// TIA Portal V19 export
FUNCTION "Route 404" : Void   // FC103, STL
TITLE = Polygon Transfer Line - CIP Sequence
{ S7_Optimized_Access := 'TRUE' }
// stored: AutoNumber false
   VAR_TEMP
      device_fault : Bool;
      switch_fault : Bool;
      tmp : Bool;
      Step_on : Bool;
      Dev_Check : Bool;
      New_Msg : Bool;
      Route_Ready : Bool;   // Ready to Run
      PNIOnodeFault : Bool;
      StepTime : S5Time;
      TimerError : Int;
      scratch_DI : DInt;
      scratch_Real : Real;
      Message : Int;
      scratch_I : Int;
      tmpWord : Word;
      PNIODiag : Struct
         node_2 : Struct
            failed : Bool;
            moduleFault : Bool;
         END_STRUCT;
         node_3 : Struct
            failed : Bool;
            moduleFault : Bool;
         END_STRUCT;
         node_4 : Struct
            failed : Bool;
            moduleFault : Bool;
         END_STRUCT;
         node_5 : Struct
            failed : Bool;
            moduleFault : Bool;
         END_STRUCT;
         node_6 : Struct
            failed : Bool;
            moduleFault : Bool;
         END_STRUCT;
         node_7 : Struct
            failed : Bool;
            moduleFault : Bool;
         END_STRUCT;
         node_8 : Struct
            failed : Bool;
            moduleFault : Bool;
         END_STRUCT;
         node_9 : Struct
            failed : Bool;
            moduleFault : Bool;
         END_STRUCT;
         node_10 : Struct
            failed : Bool;
            moduleFault : Bool;
            node_10 : Struct
               failed : Bool;
               moduleFault : Bool;
            END_STRUCT;
            node_11 : Struct
               failed : Bool;
               moduleFault : Bool;
               node_10 : Struct
                  failed : Bool;
                  moduleFault : Bool;
               END_STRUCT;
            END_STRUCT;
         END_STRUCT;
         node_11 : Struct
            failed : Bool;
            moduleFault : Bool;
            node_10 : Struct
               failed : Bool;
               moduleFault : Bool;
            END_STRUCT;
         END_STRUCT;
         node_12 : Struct
            failed : Bool;
            moduleFault : Bool;
            node_10 : Struct
               failed : Bool;
               moduleFault : Bool;
            END_STRUCT;
         END_STRUCT;
      END_STRUCT;
      TV_above_zero : Bool;
      TV_equal_zero : Bool;
      __PlcmigTempFillBit_38B2 : Bool;
      __PlcmigTempFillBit_38B3 : Bool;
      __PlcmigTempFillBit_38B4 : Bool;
      __PlcmigTempFillBit_38B5 : Bool;
      __PlcmigTempFillBit_38B6 : Bool;
      __PlcmigTempFillBit_38B7 : Bool;
      __PlcmigTempFillBit_39B0 : Bool;
      __PlcmigTempFillBit_39B1 : Bool;
      __PlcmigTempFillBit_39B2 : Bool;
      __PlcmigTempFillBit_39B3 : Bool;
      __PlcmigTempFillBit_39B4 : Bool;
      __PlcmigTempFillBit_39B5 : Bool;
      __PlcmigTempFillBit_39B6 : Bool;
      __PlcmigTempFillBit_39B7 : Bool;
   END_VAR
BEGIN

NETWORK
TITLE = PNIO 100 Node Faults
// PNIO Node 2
// PNIO Node 2
      A     "Module Diagnostic Result"."2_AL1103".ErrorValue.%X1;
      =     #PNIODiag.node_2.failed;
      A     "Module Diagnostic Result"."2_AL1103".ErrorValue.%X2;
      =     #PNIODiag.node_2.moduleFault;
// PNIO Node 3
      A     "Module Diagnostic Result"."3_AL1307".ErrorValue.%X1;
      =     #PNIODiag.node_3.failed;
      A     "Module Diagnostic Result"."3_AL1307".ErrorValue.%X2;
      =     #PNIODiag.node_3.moduleFault;
// PNIO Node 4
      A     "Module Diagnostic Result"."4_AL1307".ErrorValue.%X1;
      =     #PNIODiag.node_4.failed;
      A     "Module Diagnostic Result"."4_AL1307".ErrorValue.%X2;
      =     #PNIODiag.node_4.moduleFault;
// PNIO Node 5
      A     "Module Diagnostic Result"."5_AL1307".ErrorValue.%X1;
      =     #PNIODiag.node_5.failed;
      A     "Module Diagnostic Result"."5_AL1307".ErrorValue.%X2;
      =     #PNIODiag.node_5.moduleFault;
// PNIO Node 6
      A     "Module Diagnostic Result"."6_AL1307".ErrorValue.%X1;
      =     #PNIODiag.node_6.failed;
      A     "Module Diagnostic Result"."6_AL1307".ErrorValue.%X2;
      =     #PNIODiag.node_6.moduleFault;
// PNIO Node 7
      A     "Module Diagnostic Result"."7_AL1307".ErrorValue.%X1;
      =     #PNIODiag.node_7.failed;
      A     "Module Diagnostic Result"."7_AL1307".ErrorValue.%X2;
      =     #PNIODiag.node_7.moduleFault;
// PNIO Node 8
      A     "Module Diagnostic Result"."8_Promag300".ErrorValue.%X1;
      =     #PNIODiag.node_8.failed;
      A     "Module Diagnostic Result"."8_Promag300".ErrorValue.%X2;
      =     #PNIODiag.node_8.moduleFault;
// PNIO Node 9
      A     "Module Diagnostic Result"."9_SinaG120".ErrorValue.%X1;
      =     #PNIODiag.node_9.failed;
      A     "Module Diagnostic Result"."9_SinaG120".ErrorValue.%X2;
      =     #PNIODiag.node_9.moduleFault;
// PNIO Node 10
      A     "Module Diagnostic Result"."10_AL1307".ErrorValue.%X1;
      =     #PNIODiag.node_10.failed;
      A     "Module Diagnostic Result"."10_AL1307".ErrorValue.%X2;
      =     #PNIODiag.node_10.moduleFault;
// PNIO Node 11
      A     "Module Diagnostic Result"."11_PNCoup".ErrorValue.%X1;
      =     #PNIODiag.node_11.failed;
      A     "Module Diagnostic Result"."11_PNCoup".ErrorValue.%X2;
      =     #PNIODiag.node_11.moduleFault;
// PNIO Node 12
      A     "Module Diagnostic Result"."12_AL1307".ErrorValue.%X1;
      =     #PNIODiag.node_12.failed;
      A     "Module Diagnostic Result"."12_AL1307".ErrorValue.%X2;
      =     #PNIODiag.node_12.moduleFault;


NETWORK
TITLE = PNIO node fault
      O     #PNIODiag.node_2.failed;
      O     #PNIODiag.node_2.moduleFault;
      O     #PNIODiag.node_3.failed;
      O     #PNIODiag.node_3.moduleFault;
      O     #PNIODiag.node_4.failed;
      O     #PNIODiag.node_4.moduleFault;
      O     #PNIODiag.node_5.failed;
      O     #PNIODiag.node_5.moduleFault;
      O     #PNIODiag.node_6.failed;
      O     #PNIODiag.node_6.moduleFault;
      O     #PNIODiag.node_7.failed;
      O     #PNIODiag.node_7.moduleFault;
      O     #PNIODiag.node_8.failed;
      O     #PNIODiag.node_8.moduleFault;
      O     #PNIODiag.node_9.failed;
      O     #PNIODiag.node_9.moduleFault;
      O     #PNIODiag.node_10.failed;
      O     #PNIODiag.node_10.moduleFault;
      O     #PNIODiag.node_11.failed;
      O     #PNIODiag.node_11.moduleFault;
      O     #PNIODiag.node_12.failed;
      O     #PNIODiag.node_12.moduleFault;
      =     #PNIOnodeFault;

NETWORK
TITLE = Device Faults
      O     "ItemAlarmsOP".Item[20];  //FB_FAULT_VALVE_09_05
      O     "ItemAlarmsOP".Item[23];  //FB_FAULT_VALVE_09_08
      O     "ItemAlarmsOP".Item[24];  //FB_FAULT_VALVE_09_09
      O     "ItemAlarmsOP".Item[25];  //FB_FAULT_VALVE_09_10
      O     "ItemAlarmsOP".Item[26];  //FB_FAULT_VALVE_09_11
      O     "ItemInfoScada".Items[68].fb_error;
      O     "ItemInfoScada".Items[69].fb_error;
      O     "ItemInfoScada".Items[70].fb_error;
      O     "ItemInfoScada".Items[85].fb_error;
      O     "ItemInfoScada".Items[71].fb_error;
      O     "ItemInfoScada".Items[72].fb_error;
      O     "ItemInfoScada".Items[73].fb_error;
      O     "ItemInfoScada".Items[74].fb_error;
      O     "ItemInfoScada".Items[78].fb_error;
      O     "ItemInfoScada".Items[79].fb_error;
      O     "ItemInfoScada".Items[80].fb_error;
      O     "ItemInfoScada".Items[81].fb_error;
      O     "ItemInfoScada".Items[82].fb_error;
      O     "ItemInfoScada".Items[83].fb_error;
      O     "ItemInfoScada".Items[75].fb_error;
      O     "ItemInfoScada".Items[76].fb_error;
      O     "ItemInfoScada".Items[77].TrippedInd;
      O     "ItemInfoScada".Items[77].IsolatedInd;
      O     "ItemInfoScada".Items[84].TrippedInd;
      O     "ItemInfoScada".Items[84].IsolatedInd;
      O     "ItemInfoScada".Items[77].fb_error;
      O     "ItemInfoScada".Items[84].fb_error;
      O     #PNIOnodeFault;
      O     "ProcessAndPbAlarms"."A"[78];  //A78_PG_PTX0940HighPress
      O     "ProcessAndPbAlarms"."A"[69];  //A69_TT0941_TempFault
      =     #device_fault;

NETWORK
TITLE = Switch Fault
      ON    "PG_Devices".DI_100_005_X06_X1_3p4;
      O     "PG_Devices".DI_100_005_X06_X1_3p2;
      O     "PG_Devices".DI_100_012_X1_1p2;
      =     #switch_fault;

NETWORK
TITLE = Set Devices in Auto
      A     "RTE_404_DB".HMI.RUNNING;
      R     "ItemInfoScada".Items[50].auto_man;
      R     "ItemInfoScada".Items[53].auto_man;
      R     "ItemInfoScada".Items[54].auto_man;
      R     "ItemInfoScada".Items[55].auto_man;
      R     "ItemInfoScada".Items[56].auto_man;
      R     "ItemInfoScada".Items[76].auto_man;
      R     "ItemInfoScada".Items[78].auto_man;
      R     "ItemInfoScada".Items[79].auto_man;
      R     "ItemInfoScada".Items[80].auto_man;
      R     "ItemInfoScada".Items[81].auto_man;
      R     "ItemInfoScada".Items[82].auto_man;
      R     "ItemInfoScada".Items[83].auto_man;
      R     "ItemInfoScada".Items[77].auto_man;
      R     "ItemInfoScada".Items[84].auto_man;

NETWORK
TITLE = Route Healthy
      AN    #device_fault;
      AN    #switch_fault;
      =     "RTE_404_DB".HMI.Route_Healthy;

NETWORK
TITLE = DEVICE FAULT STATUS
      A     #device_fault;
      AN    "RTE_404_TestBit";
      =     "RTE_404_DB".FLAGS.Device_Fault;

NETWORK
TITLE = GENERAL FAULT STATUS
      O     #switch_fault;
      O     "RTE_404_DB".FLAGS.Device_Fault;
      A     "RTE_404_DB".HMI.RUNNING;
      =     "RTE_404_DB".HMI.FAULT;

NETWORK
TITLE = Temporary Message Store
// Clear down temporary message store.
      L     0;
      T     #Message;
      NOP   0;

NETWORK
TITLE = Generate Sequence Start Command
// The sequence is initiated via the interface signals ..afl
      A     "RTE_404_DB".HMI_CMD.Start;
      AN    "RTE_404_DB".HMI.RUNNING;
      A     "RTE_404_DB".HMI.Route_Healthy;
      =     "RTE_404_DB".FLAGS.Sequence_Start;


      A     "RTE_404_DB".HMI_CMD.Start;
      A     "RTE_404_DB".HMI.SEQUENCE_ABORTED;
      JCN   a10a;
      L     0;
      T     "RTE_404_DB".HMI.NEXT_STEP;
a10a: NOP   0;

      AN    "RTE_404_DB".HMI.RUNNING;
      A     "RTE_404_DB".HMI.Route_Healthy;
      =     "RTE_404_DB".HMI_CMD.Start_Available;


NETWORK
TITLE = ****ERROR MESSAGE****
// Message 10 - Device Fault
      A(;
      O     "RTE_404_DB".HMI_CMD.Start;
      O     "RTE_404_DB".HMI_CMD.Continue;
      );
      A     #device_fault;
      JNB   _001;
      L     10;
      T     #Message;
      SET;
      SAVE;
      CLR;
_001: A     BR;
      JC    AA01;

NETWORK
TITLE = ****ERROR MESSAGE****
// Message 12 - Control Stop activated
      A(;
      O     "RTE_404_DB".HMI_CMD.Start;
      O     "RTE_404_DB".HMI_CMD.Continue;
      );
      A(;
      O     "PG_Devices".DI_100_012_X1_1p2;
      O;
      A     "RTE_404_DB".FLAGS.STEP_4_0;
      AN    "CIP_Running";
      );
      JNB   _002;
      L     41;
      T     #Message;
      SET;
      SAVE;
      CLR;
_002: A     BR;
      JC    AA01;

NETWORK
TITLE = ****ERROR MESSAGE****
// Message 37 - Swingbend out of position
      A(;
      O     "RTE_404_DB".HMI_CMD.Start;
      O     "RTE_404_DB".HMI_CMD.Continue;
      );
      A(;
      O     "PG_Devices".DI_100_005_X06_X1_3p2;
      ON    "PG_Devices".DI_100_005_X06_X1_3p4;
      );
      JNB   _003;
      L     37;
      T     #Message;
      SET;
      SAVE;
      CLR;
_003: A     BR;
      JC    AA01;

NETWORK
TITLE = ****ERROR MESSAGE****
// Message 17 - Sequence Not Held
// To abort or continue the clean it must have already been held.
      A(;
      O     "RTE_404_DB".HMI_CMD.Abort;
      O     "RTE_404_DB".HMI_CMD.Continue;
      );
      AN    "RTE_404_DB".HMI.SEQUENCE_HELD;
      JNB   _004;
      L     17;
      T     #Message;
      SET;
      SAVE;
      CLR;
_004: A     BR;
      JC    AA01;

NETWORK
TITLE = ****ERROR MESSAGE****
// Message 21 - Line Sterilising
// *** Use Sterilising Seq running bit ***
      A(;
      O     "RTE_404_DB".HMI_CMD.Start;
      O     "RTE_404_DB".HMI_CMD.Continue;
      );
      A     "ATI";
      AN    "ATI";
      JNB   _005;
      L     21;
      T     #Message;
      SET;
      SAVE;
      CLR;
_005: A     BR;
      JC    AA01;

NETWORK
TITLE = ****ERROR MESSAGE****
// Message 22 - Inhibited by Running Sequence
// *** Use Production Seq running bit ***
      A(;
      O     "RTE_404_DB".HMI_CMD.Start;
      O     "RTE_404_DB".HMI_CMD.Continue;
      );
      A(;
      O     "RTE_405_DB".HMI.RUNNING;
      O     "RTE_406_DB".HMI.RUNNING;
      );
      JNB   _006;
      L     22;
      T     #Message;
      SET;
      SAVE;
      CLR;
_006: A     BR;
      JC    AA01;

NETWORK
TITLE = ****ERROR MESSAGE****
// Message 25 - CIP Not Running
      A(;
      O     "RTE_404_DB".HMI_CMD.Start;
      O     "RTE_404_DB".HMI_CMD.Continue;
      );
      A     "RTE_404_DB".FLAGS.STEP_4_0;
      AN    "CIP_Running";
      JNB   _007;
      L     25;
      T     #Message;
      SET;
      SAVE;
      CLR;
_007: A     BR;
      JC    AA01;

NETWORK
TITLE = New Message Detected
AA01: A(;
      L     #Message;
      L     0;
      <>I;
      );
      JNB   _008;
      L     #Message;
      T     "RTE_404_DB".HMI.ERROR_TEXT_NUMBER;
      SET;
      SAVE;
      CLR;
_008: A     BR;
      =     #New_Msg;

NETWORK
TITLE = ****NEW ERROR MESSAGE****
// Reset all CIP commands except START.
// On a new non-zero error message being displayed reset all commands from SCADA 
// so they take no action. Also, start a delay off timer to cancel display of the 
// error message.
      A     #New_Msg;
      R     "RTE_404_DB".HMI_CMD.Abort;
      R     "RTE_404_DB".HMI_CMD.Continue;
      R     "RTE_404_DB".HMI_CMD.Hold;
      R     "RTE_404_DB".HMI_CMD.Timer_Release;
      R     "RTE_404_DB".HMI_CMD.Timer_Hold;
      R     "RTE_404_DB".FLAGS.Sequence_Start;
      L     S5T#10S;
      SF    "RTE404_MSG";

NETWORK
TITLE = ****NEW ERROR MESSAGE****
// Error message display cancel.
      AN    "RTE404_MSG";
      JNB   _009;
      L     0;
      T     "RTE_404_DB".HMI.ERROR_TEXT_NUMBER;
_009: NOP   0;

NETWORK
TITLE = ROUTE RUNNING
      L     "RTE_404_DB".HMI.STEP_NUMBER;
      L     0;
      <>I;
      =     "RTE_404_DB".HMI.RUNNING;

NETWORK
TITLE = ****SEQ ABORT****
      A     "RTE_404_DB".HMI_CMD.Abort;
      A     "RTE_404_DB".HMI.SEQUENCE_HELD;
      S     "RTE_404_DB".HMI.SEQUENCE_ABORTED;

      A     "RTE_404_DB".HMI.SEQUENCE_HELD;
      =     "RTE_404_DB".HMI_CMD.Abort_Available;


NETWORK
TITLE = Enable HMI Hold Pb
      A     "RTE_404_DB".HMI.RUNNING;
      =     "RTE_404_DB".HMI_CMD.Hold_Available;

NETWORK
TITLE = Sequence held flag
// Set sequence hold if sequence is running and a hold fault condition is detected 
// or a sequence hold command is received from SCADA.
// 
// When a validated CONTINUE command is received from SCADA and all fault 
// conditions are cleared then reset sequence hold.
// 
// Added "Product Request" (CIP Complete) to prevent sequence going into hold when 
// Central CIP completes
      A(;
      O     "RTE_404_DB".HMI_CMD.Hold;
      ON    "RTE_404_DB".HMI.Route_Healthy;
      O;
      A(;
      O     "RTE_404_DB".FLAGS.STEP_3_0;
      O     "RTE_404_DB".FLAGS.STEP_4_0;
      );
      AN    "Product_Request";
      AN    "CIP_Running";
      );
      A     "RTE_404_DB".HMI.RUNNING;
      =     #__PlcmigTempFillBit_39B0;
      A     #__PlcmigTempFillBit_39B0;
      BLD   102;
      S     "RTE_404_DB".HMI.SEQUENCE_HELD;
      A     #__PlcmigTempFillBit_39B0;
      NOT;
      =     #__PlcmigTempFillBit_39B1;
      A     #__PlcmigTempFillBit_39B1;
      A(;
      O     "RTE_404_DB".HMI_CMD.Continue;
      O     "RTE_404_DB".HMI_CMD.Abort;
      );
      R     "RTE_404_DB".HMI.SEQUENCE_HELD;
      A     #__PlcmigTempFillBit_39B1;
      A     "RTE_404_DB".HMI.SEQUENCE_HELD;
      =     "RTE_404_DB".HMI_CMD.Continue_Available;

NETWORK
TITLE = Sequence held flag
// Reset when circuit not running i.e after an abort.
      A     "RTE_404_DB".FLAGS.STEP_0;
      AN    "RTE_404_DB".HMI.RUNNING;
      R     "RTE_404_DB".HMI.SEQUENCE_HELD;

NETWORK
TITLE = ****RESET ABORT FLAG****
      A     "RTE_404_DB".FLAGS.STEP_0;
      A     "RTE_404_DB".FLAGS.Step_Change;
      R     "RTE_404_DB".HMI.SEQUENCE_ABORTED;

NETWORK
TITLE = Step 0.0 Reset
      AN    "RTE_404_DB".HMI.RUNNING;
      AN    "RTE_404_DB".FLAGS.STEP_0;
      =     #Step_on;

NETWORK
TITLE = Step 0.0 Reset
// Reset sequnece to step 0 and clear down step value and dimension words.
      A(;
      A(;
      A(;
      O     #Step_on;
      O;
      A     "RTE_404_DB".FLAGS.STEP_0;
      A     "RTE_404_DB".FLAGS.Step_Change;
      );
      JNB   _00a;
      L     0;
      T     "RTE_404_DB".HMI.NEXT_STEP;
      SET;
      SAVE;
      CLR;
_00a: A     BR;
      );
      JNB   _00b;
      L     0;
      T     "RTE_404_DB".HMI.STEP_VALUE;
      SET;
      SAVE;
      CLR;
_00b: A     BR;
      );
      JNB   _00c;
      L     0;
      T     "RTE_404_DB".HMI.STEP_VALUE_DIMENSION;
_00c: NOP   0;

NETWORK
TITLE = Move to Step 0.5
      A     "RTE_404_DB".FLAGS.STEP_0;
      A     "RTE_404_DB".FLAGS.Sequence_Start;
      =     #__PlcmigTempFillBit_39B0;
      A     #__PlcmigTempFillBit_39B0;
      BLD   102;
      =     #Step_on;
      A     #__PlcmigTempFillBit_39B0;
      JNB   _00d;
      L     5;
      T     "RTE_404_DB".HMI.NEXT_STEP;
_00d: NOP   0;

NETWORK
TITLE = Set Line Status Unsterile
      A     #Step_on;
      R     "RTE_404_DB".FLAGS.Clean;
      R     "RTE_405_DB".FLAGS.Sterile;

NETWORK
TITLE = Move to Step 1.0
      A(;
      L     "RTE_404_DB".HMI.NEXT_STEP;
      L     5;
      ==I;
      );
      A     "CIP_Route_Request";
      AN    "RTE_404_DB".FLAGS.Step_Change;
      =     #__PlcmigTempFillBit_39B0;
      A     #__PlcmigTempFillBit_39B0;
      BLD   102;
      =     #Step_on;
      A     #__PlcmigTempFillBit_39B0;
      JNB   _00e;
      L     10;
      T     "RTE_404_DB".HMI.NEXT_STEP;
_00e: NOP   0;

NETWORK
TITLE = Dev Check
// Dev Check following Route valves Open - 09.10, 09.08, 09.45, 10.21, 10.23, 10.25
// and following Route Valves closed - 09.09, 09.05, 10.24
      A     "RTE_404_DB".FLAGS.STEP_1_0;
      A     "Y0905R";
      A     "Y0908S";
      A     "Y0909R";
      A     "Y0910S";
      A(;
      A     "ItemInfoScada".Items[78].Set_FB;
      A     "ItemInfoScada".Items[79].Set_FB;
      A     "ItemInfoScada".Items[80].Reset_FB;
      );
      =     #Dev_Check;

NETWORK
TITLE = Move to Step 2.0
      A     "RTE_404_DB".FLAGS.STEP_1_0;
      A     #Dev_Check;
      AN    "RTE_404_DB".FLAGS.Step_Change;
      =     #__PlcmigTempFillBit_39B0;
      A     #__PlcmigTempFillBit_39B0;
      BLD   102;
      =     #Step_on;
      A     #__PlcmigTempFillBit_39B0;
      JNB   _00f;
      L     20;
      T     "RTE_404_DB".HMI.NEXT_STEP;
_00f: NOP   0;

NETWORK
TITLE = Check Condenstate OK, then Set CIP Route Open
      A     "RTE_404_DB".FLAGS.STEP_2_0;
      A     "CIP_Route_Request";
      A     "M21.2";
      S     "RTE_404_Cip_Route_Open";

NETWORK
TITLE = Move to Step 3.0
      A     "RTE_404_DB".FLAGS.STEP_2_0;
      A     "CIP_Running";
      AN    "RTE_404_DB".FLAGS.Step_Change;
      =     #__PlcmigTempFillBit_39B0;
      A     #__PlcmigTempFillBit_39B0;
      BLD   102;
      =     #Step_on;
      A     #__PlcmigTempFillBit_39B0;
      JNB   _010;
      L     30;
      T     "RTE_404_DB".HMI.NEXT_STEP;
_010: NOP   0;

NETWORK
TITLE = Reset Totaliser Value
// Totaliser Control
// 0 = Totalise
// 3 = Reset + Totalise
      O(;
      A(;
      A(;
      O     "RTE_404_DB".FLAGS.STEP_3_0;
      O;
      AN    "M21.2";
      A     "RTE_404_DB".FLAGS.STEP_4_0;
      );
      =     "RTE_404_Sip_Steam";
      A     "RTE_404_Sip_Steam";
      JNB   _011;
      L     "RTE_404_DB".PARAMETERS.PARAM_01;
      ITD;
      T     #scratch_DI;
      SET;
      SAVE;
      CLR;
_011: A     BR;
      );
      JNB   _012;
      L     #scratch_DI;
      DTR;
      T     #scratch_Real;
      SET;
      SAVE;
      CLR;
_012: A     BR;
      );
      O(;
      A(;
      O     #Step_on;
      O;
      A     "RTE_404_DB".FLAGS.STEP_3_0;
      A(;
      O     #device_fault;
      ON    "CIP_Running";
      );
      );
      A(;
      L     "PG_Devices".FT0940.Totaliser_Value;
      L     0.0;
      <>R;
      );
      =     #TV_above_zero;
      A     #TV_above_zero;
      JNB   _013;
      L     1;
      T     "PG_Devices".FT0940.Totaliser_Control;
      SET;
      SAVE;
      CLR;
_013: A     BR;
      );
      O(;
      A(;
      A     "RTE_404_DB".FLAGS.STEP_3_0;
      A(;
      L     "PG_Devices".FT0940.Totaliser_Value;
      L     0.0;
      <=R;
      );
      JNB   _014;
      L     0;
      T     "PG_Devices".FT0940.Totaliser_Control;
      SET;
      SAVE;
      CLR;
_014: A     BR;
      );
      =     #TV_equal_zero;
      A     #TV_equal_zero;
      );
      O(;
      A     #TV_above_zero;
      S     "RTE_404_DB".FLAGS.TotaliserResetBit;
      A     #TV_equal_zero;
      R     "RTE_404_DB".FLAGS.TotaliserResetBit;
      A     "RTE_404_DB".FLAGS.TotaliserResetBit;
      );
      =     #tmp;

NETWORK
TITLE = Move to Step 4.0
      AN    "RTE_404_DB".FLAGS.TotaliserResetBit;
      A     "RTE_404_DB".FLAGS.STEP_3_0;
      A(;
      L     "PG_Devices".FT0940.Totaliser_Value;
      L     #scratch_Real;
      >=R;
      );
      AN    "RTE_404_DB".FLAGS.Step_Change;
      =     #__PlcmigTempFillBit_39B0;
      A     #__PlcmigTempFillBit_39B0;
      BLD   102;
      =     #Step_on;
      A     #__PlcmigTempFillBit_39B0;
      JNB   _015;
      L     40;
      T     "RTE_404_DB".HMI.NEXT_STEP;
_015: NOP   0;

NETWORK
TITLE = EOL Valve Flips Interval Timer
      A     "RTE_404_DB".FLAGS.STEP_4_0;
      AN    "RTE_404_DB".FLAGS.ENCYL_3;
      AN    "RTE_404_DB".HMI.SEQUENCE_HELD;
      =     #__PlcmigTempFillBit_39B0;
      BLD   103;
      A     "RTE_404_DB".FLAGS.ENCYL_3;
      =     #__PlcmigTempFillBit_39B1;
      BLD   103;
      A(;
      A(;
      L     "RTE_404_DB".PARAMETERS.PARAM_03;
      ITD;
      T     #scratch_DI;
      SET;
      SAVE;
      CLR;
      A     BR;
      );
      JNB   _016;
      L     #scratch_DI;
      L     1000;
      *D;
      T     #scratch_DI;
      AN    OV;
      SAVE;
      CLR;
_016: A     BR;
      );
      JNB   _017;
      CALL  "TONR"
      ( TMR_EN  := #__PlcmigTempFillBit_39B0,
        RESET   := #__PlcmigTempFillBit_39B1,
        PV      := #scratch_DI,
        DELTA_T := "Last Scan Time",
        Q       := "RTE_404_DB".FLAGS.ENCYL_1,
        ET      := "RTE_404_DB".PARAMETERS.PARAM_03_Act
      );
_017: NOP   0;

NETWORK
TITLE = Cycle 1 to Cycle 2 Delay Timer.
      A     "RTE_404_DB".FLAGS.STEP_4_0;
      A     "RTE_404_DB".FLAGS.ENCYL_1;
      AN    "RTE_404_DB".HMI.SEQUENCE_HELD;
      =     #__PlcmigTempFillBit_39B0;
      BLD   103;
      AN    "RTE_404_DB".FLAGS.ENCYL_1;
      =     #__PlcmigTempFillBit_39B1;
      BLD   103;
      A(;
      A(;
      L     "RTE_404_DB".PARAMETERS.PARAM_04;
      ITD;
      T     #scratch_DI;
      SET;
      SAVE;
      CLR;
      A     BR;
      );
      JNB   _018;
      L     #scratch_DI;
      L     1000;
      *D;
      T     #scratch_DI;
      AN    OV;
      SAVE;
      CLR;
_018: A     BR;
      );
      JNB   _019;
      CALL  "TONR"
      ( TMR_EN  := #__PlcmigTempFillBit_39B0,
        RESET   := #__PlcmigTempFillBit_39B1,
        PV      := #scratch_DI,
        DELTA_T := "Last Scan Time",
        Q       := "RTE_404_DB".FLAGS.ENCYL_2,
        ET      := "RTE_404_DB".PARAMETERS.PARAM_04_Act
      );
_019: NOP   0;

NETWORK
TITLE = Cycle 2 to Cycle 3 Overlapping Timers.
      A     "RTE_404_DB".FLAGS.STEP_4_0;
      A     "RTE_404_DB".FLAGS.ENCYL_2;
      =     #__PlcmigTempFillBit_39B0;
      A     #__PlcmigTempFillBit_39B0;
      L     S5T#2S;
      SD    "Tag_78";
      NOP   0;
      NOP   0;
      NOP   0;
      NOP   0;
      A     #__PlcmigTempFillBit_39B0;
      BLD   102;
      L     S5T#2S;
      SF    "T83";

NETWORK
TITLE = Cycle 2 + T69 (2 Secs) to Cycle 3 Delay Timer.
      A     "RTE_404_DB".FLAGS.STEP_4_0;
      A     "RTE_404_DB".FLAGS.ENCYL_2;
      A     "Tag_78";
      AN    "RTE_404_DB".HMI.SEQUENCE_HELD;
      =     #__PlcmigTempFillBit_39B0;
      BLD   103;
      AN    "RTE_404_DB".FLAGS.ENCYL_2;
      =     #__PlcmigTempFillBit_39B1;
      BLD   103;
      A(;
      A(;
      L     "RTE_404_DB".PARAMETERS.PARAM_05;
      ITD;
      T     #scratch_DI;
      SET;
      SAVE;
      CLR;
      A     BR;
      );
      JNB   _01a;
      L     #scratch_DI;
      L     1000;
      *D;
      T     #scratch_DI;
      AN    OV;
      SAVE;
      CLR;
_01a: A     BR;
      );
      JNB   _01b;
      CALL  "TONR"
      ( TMR_EN  := #__PlcmigTempFillBit_39B0,
        RESET   := #__PlcmigTempFillBit_39B1,
        PV      := #scratch_DI,
        DELTA_T := "Last Scan Time",
        Q       := "RTE_404_DB".FLAGS.ENCYL_3,
        ET      := "RTE_404_DB".PARAMETERS.PARAM_05_Act
      );
_01b: NOP   0;

NETWORK
TITLE = Move to Step 5.0
// Product_Request means "CIP Complete" in this context.
      A(;
      A     "RTE_404_DB".FLAGS.STEP_4_0;
      A     "Product_Request";
      O;
      A     "RTE_404_DB".HMI_CMD.Abort;
      A     "RTE_404_DB".HMI.SEQUENCE_ABORTED;
      );
      AN    "RTE_404_DB".FLAGS.Step_Change;
      =     #__PlcmigTempFillBit_39B0;
      A     #__PlcmigTempFillBit_39B0;
      BLD   102;
      =     #Step_on;
      A     #__PlcmigTempFillBit_39B0;
      JNB   _01c;
      L     50;
      T     "RTE_404_DB".HMI.NEXT_STEP;
_01c: NOP   0;

NETWORK
TITLE = Move to Step 6.0
      A     "RTE_404_DB".FLAGS.STEP_5_0;
      A     "Y0910R";
      =     #__PlcmigTempFillBit_39B0;
      A     #__PlcmigTempFillBit_39B0;
      AN    "RTE_404_DB".FLAGS.Step_Change;
      =     #__PlcmigTempFillBit_39B1;
      A     #__PlcmigTempFillBit_39B1;
      BLD   102;
      =     #Step_on;
      A     #__PlcmigTempFillBit_39B1;
      JNB   _01d;
      L     60;
      T     "RTE_404_DB".HMI.NEXT_STEP;
_01d: NOP   0;
      A     #__PlcmigTempFillBit_39B0;
      BLD   102;
      R     "RTE_404_Cip_Route_Open";

NETWORK
TITLE = Dev Check
// Check following valve are open  V09.11, V10.25, V10.27, V10.83
      A     "RTE_404_DB".FLAGS.STEP_6_0;
      A     "Y0908S";
      A     "Y0910R";
      A     "Y0911S";
      A(;
//   A     "ItemInfoScada".items[79].Set_FB
      A     "ItemInfoScada".Items[81].Set_FB;
      A     "ItemInfoScada".Items[82].Set_FB;
      A     "ItemInfoScada".Items[83].Set_FB;
      );
      =     #Dev_Check;

NETWORK
TITLE = Move to Step 7.0
      A     "RTE_404_DB".FLAGS.STEP_6_0;
      A     #Dev_Check;
      AN    "RTE_404_DB".FLAGS.Step_Change;
      =     #__PlcmigTempFillBit_39B0;
      A     #__PlcmigTempFillBit_39B0;
      BLD   102;
      =     #Step_on;
      A     #__PlcmigTempFillBit_39B0;
      JNB   _01e;
      L     70;
      T     "RTE_404_DB".HMI.NEXT_STEP;
_01e: NOP   0;

NETWORK
TITLE = Initialise Step Parameters
      A(;
      A     #Step_on;
      JNB   _01f;
      L     "RTE_404_DB".PARAMETERS.PARAM_02;
      T     "RTE_404_DB".HMI.STEP_VALUE;
      SET;
      SAVE;
      CLR;
_01f: A     BR;
      );
      JNB   _020;
      L     1;
      T     "RTE_404_DB".HMI.STEP_VALUE_DIMENSION;
_020: NOP   0;

NETWORK
TITLE = Move to Step 8.0
      A     "RTE_404_DB".FLAGS.STEP_7_0;
      A     "RTE_404_DB".FLAGS.Step_Value_Done;
      AN    "RTE_404_DB".FLAGS.Step_Change;
      =     #__PlcmigTempFillBit_39B0;
      A     #__PlcmigTempFillBit_39B0;
      BLD   102;
      =     #Step_on;
      A     #__PlcmigTempFillBit_39B0;
      JNB   _021;
      L     80;
      T     "RTE_404_DB".HMI.NEXT_STEP;
_021: NOP   0;

NETWORK
TITLE = Dev Check
// V09.11
//     V09.08
//     V10.21
//     V10.23
//     V10.27
//     V10.83
//     V10.25
      A     "Y0908R";
      A     "Y0911R";
      A     "ItemInfoScada".Items[78].Reset_FB;
      A     "ItemInfoScada".Items[79].Reset_FB;
      A     "ItemInfoScada".Items[81].Reset_FB;
      A     "ItemInfoScada".Items[82].Reset_FB;
      A     "ItemInfoScada".Items[83].Reset_FB;
      =     #Dev_Check;

NETWORK
TITLE = Move to Step END
      A     "RTE_404_DB".FLAGS.STEP_8_0;
      A     #Dev_Check;
      AN    "RTE_404_DB".FLAGS.Step_Change;
      =     #__PlcmigTempFillBit_39B0;
      A     #__PlcmigTempFillBit_39B0;
      BLD   102;
      =     #Step_on;
      A     #__PlcmigTempFillBit_39B0;
      JNB   _022;
      L     90;
      T     "RTE_404_DB".HMI.NEXT_STEP;
_022: NOP   0;

NETWORK
TITLE = Set Line Status Unsterile
      A     #Step_on;
      AN    "RTE_404_DB".HMI.SEQUENCE_ABORTED;
      S     "RTE_404_DB".FLAGS.Clean;

NETWORK
TITLE = Move to Step 0.0
      A     "RTE_404_DB".FLAGS.STEP_END;
      A     "RTE_404_DB".FLAGS.Step_Value_Done;
      AN    "RTE_404_DB".FLAGS.Step_Change;
      =     #__PlcmigTempFillBit_39B0;
      A     #__PlcmigTempFillBit_39B0;
      BLD   102;
      =     #Step_on;
      A     #__PlcmigTempFillBit_39B0;
      JNB   _023;
      L     0;
      T     "RTE_404_DB".HMI.NEXT_STEP;
_023: NOP   0;

NETWORK
TITLE = Step Change Detected
// The next step number is different to the current step then set flag.
      L     "RTE_404_DB".HMI.NEXT_STEP;
      L     "RTE_404_DB".HMI.STEP_NUMBER;
      <>I;
      =     "RTE_404_DB".FLAGS.Step_Change;

NETWORK
TITLE = Current step value decremented to zero
      A(;
      L     "RTE_404_DB".HMI.STEP_VALUE;
      L     0;
      <=I;
      );
      AN    "RTE_404_DB".FLAGS.Step_Change;
      =     "RTE_404_DB".FLAGS.Step_Value_Done;

NETWORK
TITLE = Enable step count down
      A(;
      A     "RTE_404_DB".FLAGS.STEP_7_0;
      A(;
      ON    "Y0908S";
      ON    "Y0910R";
      ON    "Y0911S";
      ON    "ItemInfoScada".Items[79].Set_FB;
      ON    "ItemInfoScada".Items[81].Set_FB;
      ON    "ItemInfoScada".Items[82].Set_FB;
      ON    "ItemInfoScada".Items[83].Set_FB;
      );
      O     "RTE_404_DB".HMI.SEQUENCE_HELD;
      );
      NOT;
      =     "RTE_404_DB".FLAGS.Step_Count_Enable;

NETWORK
TITLE = Decrement Step Value
// With count enabled and timer not held count down on each 1 second pulse.
      A     "RTE_404_DB".HMI.RUNNING;
      A     "RTE_404_DB".FLAGS.Step_Count_Enable;
      AN    "RTE_404_DB".HMI.TIMER_HELD;
      AN    "RTE_404_DB".FLAGS.Step_Value_Done;
      A     "1HZ_ONESHOT";
      JNB   _024;
      L     "RTE_404_DB".HMI.STEP_VALUE;
      L     1;
      -I;
      T     "RTE_404_DB".HMI.STEP_VALUE;
_024: NOP   0;

NETWORK
TITLE = Reset HMI commands
      A     "ATI";
      R     "RTE_404_DB".HMI_CMD.Abort;
      R     "RTE_404_DB".HMI_CMD.Continue;
      R     "RTE_404_DB".HMI_CMD.Hold;
      R     "RTE_404_DB".HMI_CMD.Timer_Release;
      R     "RTE_404_DB".HMI_CMD.Timer_Hold;
      R     "RTE_404_DB".HMI_CMD.Start;

NETWORK
TITLE = MESSAGE CLEARANCE TIMING
      A     "1HZ_ONESHOT";
      =     #__PlcmigTempFillBit_39B0;
      BLD   103;
      CALL  "ERROR_MSG_CLEAR"
      ( MESSAGE_CLEAR_TIME := 10,
        SECOND_PULSE       := #__PlcmigTempFillBit_39B0,
        ERROR_MESSAGE      := "RTE_404_DB".HMI.ERROR_TEXT_NUMBER,
        ERROR_MESSAGE_MEM  := "RTE_404_DB".CONTROL.ERROR_MESSAGE_MEM,
        ELAPSED_TIME       := "RTE_404_DB".CONTROL.MESSAGE_TIME
      );
      NOP   0;

NETWORK
TITLE = STEP TIMER
// On detection of a new step, the timer is reset to 0 and will then start timing 
// whilst on the current step.
      A     "1HZ_ONESHOT";
      =     #__PlcmigTempFillBit_39B0;
      BLD   103;
      CALL  "STEP_TIMER"
      ( DBNR                   := 404,
        NEXT_STEP_LOCATION     := 18,
        STEP_NUM_LOCATION      := 2,
        TIME_PULSE             := #__PlcmigTempFillBit_39B0,
        STEP_TIME_ACC_LOCATION := 26
      );
      NOP   0;

NETWORK
TITLE = 
      A     "RTE_404_DB".FLAGS.Step_Change;
      JNB   _025;
      L     "RTE_404_DB".HMI.NEXT_STEP;
      T     "RTE_404_DB".HMI.STEP_NUMBER;
_025: NOP   0;

NETWORK
TITLE = Spare
      L     "RTE_404_DB".HMI.STEP_NUMBER;
      L     0;
      ==I;
      =     "RTE_404_DB".FLAGS.STEP_0;

NETWORK
TITLE = Spare
      O     "RTE_404_DB".HMI.RUNNING;
      ON    "RTE_404_DB".HMI.RUNNING;
      =     #__PlcmigTempFillBit_39B0;
      A     #__PlcmigTempFillBit_39B0;
      A(;
      L     "RTE_404_DB".HMI.STEP_NUMBER;
      L     10;
      ==I;
      );
      =     "RTE_404_DB".FLAGS.STEP_1_0;
      A     #__PlcmigTempFillBit_39B0;
      A(;
      L     "RTE_404_DB".HMI.STEP_NUMBER;
      L     20;
      ==I;
      );
      =     "RTE_404_DB".FLAGS.STEP_2_0;
      A     #__PlcmigTempFillBit_39B0;
      A(;
      L     "RTE_404_DB".HMI.STEP_NUMBER;
      L     30;
      ==I;
      );
      =     "RTE_404_DB".FLAGS.STEP_3_0;
      A     #__PlcmigTempFillBit_39B0;
      A(;
      L     "RTE_404_DB".HMI.STEP_NUMBER;
      L     40;
      ==I;
      );
      =     "RTE_404_DB".FLAGS.STEP_4_0;
      A     #__PlcmigTempFillBit_39B0;
      A(;
      L     "RTE_404_DB".HMI.STEP_NUMBER;
      L     50;
      ==I;
      );
      =     "RTE_404_DB".FLAGS.STEP_5_0;
      A     #__PlcmigTempFillBit_39B0;
      A(;
      L     "RTE_404_DB".HMI.STEP_NUMBER;
      L     60;
      ==I;
      );
      =     "RTE_404_DB".FLAGS.STEP_6_0;
      A     #__PlcmigTempFillBit_39B0;
      A(;
      L     "RTE_404_DB".HMI.STEP_NUMBER;
      L     70;
      ==I;
      );
      =     "RTE_404_DB".FLAGS.STEP_7_0;
      A     #__PlcmigTempFillBit_39B0;
      A(;
      L     "RTE_404_DB".HMI.STEP_NUMBER;
      L     80;
      ==I;
      );
      =     "RTE_404_DB".FLAGS.STEP_8_0;
      A     #__PlcmigTempFillBit_39B0;
      A(;
      L     "RTE_404_DB".HMI.STEP_NUMBER;
      L     90;
      >=I;
      );
      =     "RTE_404_DB".FLAGS.STEP_END;

NETWORK
TITLE = COPY CURRENT STEP TO STEP TEXT WORD
      L     "RTE_404_DB".HMI.STEP_NUMBER;
      T     "RTE_404_DB".HMI.STEP_IDENT_TEXT_NUMBER;
      NOP   0;
END_FUNCTION
